Staubli VAL3: libGeneric_0_1.dtx

mdesc mNomSpeed
